{attribute 'hide_all_locals'}
FUNCTION_BLOCK ResetGroup EXTENDS TaskBase
VAR_INPUT
END_VAR
VAR_OUTPUT
END_VAR
VAR
	groupReset			: MC_GroupReset;
	_caGroup			: ICollisionGroup;
	_resetGroup : BOOL;
	Logger : TcMessage_Ext;
END_VAR

CASE State OF
	0:
		IF _resetGroup THEN
			_done := FALSE;
			_error := FALSE;
			_busy := TRUE;
			groupReset.Execute := TRUE;
			IF groupReset.Busy THEN
				State := 10;
				_resetGroup := FALSE;
				Logger.Send(TC_EVENTS.XtsCAGroupEvents.CAGroupResetting,'');
			END_IF
		END_IF
	
	10:
		IF NOT groupReset.Busy THEN
			IF groupReset.Done THEN
				_done := TRUE;
				Logger.Send(TC_EVENTS.XtsCAGroupEvents.CAGroupResetDone,'');
			ELSIF groupReset.Error THEN
				_error := TRUE;
				Logger.Send(TC_EVENTS.XtsCAGroupEvents.CAGroupResetError,'');
			END_IF
			_busy := FALSE;
			groupReset.Execute := false;
			State := 0;
		END_IF
END_CASE


groupReset(AxesGroup := _caGroup.GroupRef);

METHOD Abort : BOOL
groupReset.Execute := FALSE;
State := 0;
Abort := true;
END_METHOD

METHOD Execute : BOOL
Execute := _resetGroup := true;
END_METHOD

METHOD FB_init : BOOL
VAR_INPUT
	bInitRetains : BOOL; // if TRUE, the retain variables are initialized (warm start / cold start)
	bInCopyCode : BOOL;  // if TRUE, the instance afterwards gets moved into the copy code (online change)
	CAGroup : ICollisionGroup;	
END_VAR
_caGroup := CAGroup;
END_METHOD

END_FUNCTION_BLOCK

(* stored: Version 1.1.0.1, ProductVersion 3.1.4024.12
   POU ResetGroup: Id {f1e61ccf-4a87-45e7-a827-c3b6233b7460}, SpecialFunc None
   Method Abort: Id {e1b95705-1b45-487a-ada9-22fe010e1325}
   Method Execute: Id {b94d2efe-3ffd-45f1-b278-c7e4c306cd7f}
   Method FB_init: Id {ca969347-dafc-49cc-a4f3-fb185af92df7} *)
